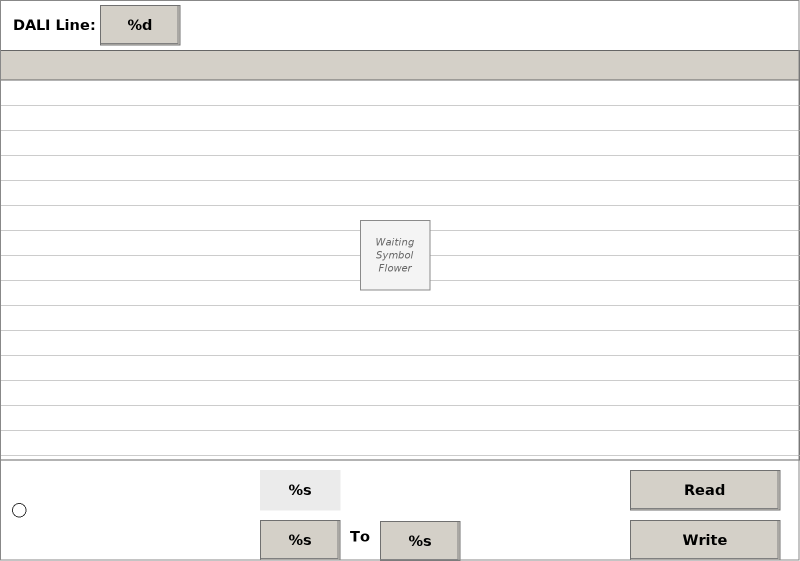
VISUALIZATION Visu_Part102Parameters  // 800x561
    Table (0,50 800x410), data array: DALI_Commissioning.fbPart102Parameters.aParameters
        p1137915858: DALI_Commissioning.fbPart102Parameters.nSelectedAddress
        p3854506369: DALI_Commissioning.fbPart102Parameters.aParameters[INDEX].nShortAddress
        p1892666644: DALI_Commissioning.fbPart102Parameters.aParameters[INDEX].nActualLevel
        p338671338: DALI_Commissioning.fbPart102Parameters.aParameters[INDEX].nMinLevel
        p2170511999: DALI_Commissioning.fbPart102Parameters.aParameters[INDEX].nMaxLevel
        p3723444502: DALI_Commissioning.fbPart102Parameters.aParameters[INDEX].eFadeRate
        p1218418051: DALI_Commissioning.fbPart102Parameters.aParameters[INDEX].eFadeTime
        p746581629: DALI_Commissioning.fbPart102Parameters.aParameters[INDEX].nPowerOnLevel
        p3104783080: DALI_Commissioning.fbPart102Parameters.aParameters[INDEX].nSystemFailureLevel
        p2501879983: DALI_Commissioning.fbPart102Parameters.aParameters[INDEX].nPhysicalMinimum
        p7306298: DALI_Commissioning.fbPart102Parameters.aParameters[INDEX].sDeviceTypes
        Columns.Column.[1].Template: OnMouseClick: write the text variable via Default, min 0, max 254, title "MinLevel"
        Columns.Column.[2].Template: OnMouseClick: write the text variable via Default, min 1, max 254, title "MaxLevel"
        Columns.Column.[3].Template: OnMouseClick: write the text variable via Default, min 0, max 254, title "FadeRate"
        Columns.Column.[4].Template: OnMouseClick: write the text variable via Default, min 1, max 15, title "Fade Rate"
        Columns.Column.[5].Template: OnMouseClick: write the text variable via Default, min 0, max 15, title "Fade Time"
        Columns.Column.[6].Template: OnMouseClick: write the text variable via Default, min 1, max 254, title "Power On Level"
        Columns.Column.[7].Template: OnMouseClick: write the text variable via Default, min 0, max 255, title "System Failure Level"
    RadioButton (10,460 254x100), variable: DALI_Commissioning.fbPart102Parameters.nAddressRange
        Areas[0]: Text=Single Short Address
        Areas[1]: Text=Short Address Range
    Textfield (335,521 50x31), "To"
    Button (630,470 150x40), "Read"
        OnMouseClick: execute { DALI_Commissioning.fbPart102Parameters.bRead := TRUE; }
    Button (630,520 150x40), "Write"
        OnMouseClick: execute { DALI_Commissioning.fbPart102Parameters.bWrite := TRUE; }
    Button (260,520 80x40), "%s", text variable: DALI_Commissioning.fbPart102Parameters.nStartAddress
        OnMouseClick: write the text variable via Default, min 0, max 63, title "Insert Short Address"
    Button (380,521 80x40), "%s", text variable: DALI_Commissioning.fbPart102Parameters.nEndAddress
        OnMouseClick: write the text variable via Default, min 0, max 63, title "Insert Short Address"
    Textfield (260,470 80x40), "%s", tooltip "Please select the desired Short Address in the table above.", text variable: DALI_Commissioning.fbPart102Parameters.nSelectedAddress
    WaitingSymbolFlower (360,220 70x70), invisible if: DALI_Commissioning.fbPart102Parameters.bHideWaitSymbol
    Group (10,5 170x40)
        Textfield (0,0 110x40), "DALI Line:"
        Button (90,0 80x40), "%d", text variable: GVL_Internal.nDALILine
            OnMouseClick: write the text variable via Default, min 1, max GVL_Internal.nNumberOfDALI_Lines, title "Choose line"
END_VISUALIZATION

(* stored: Version 1.1.0.1, ProductVersion 3.1.4024.12
   Visu Visu_Part102Parameters: Id {78b18f00-7947-4538-8cdc-09981442750e} *)
